FUNCTION_BLOCK FB_A_Magnetventil IMPLEMENTS I_Magnetventil
VAR_INPUT
	I_iModus			:INT;		// Zustand des Systems (z.B. 0 = AUS | 1 = MAN | 2 = AUTO)
	I_bVerriegeln		:BOOL;		// Verriegelte Elemente sind nicht ansteuerbar
END_VAR

VAR_OUTPUT
	O_bAktivieren		:BOOL;		// Ventil wird geöffnet / geschlossen
	O_bStoerung			:BOOL;		// Befindet sich das Element in einem Error
	O_iStoerungID		:INT;		// Anzeigen von Störung über eine INT-Variable
END_VAR

VAR
END_VAR

// Verriegeln des Systems (Element geht in definierten Zustand) -> Ventil wird geschlossen
IF I_bVerriegeln THEN
	O_bAktivieren := FALSE;
END_IF

METHOD M_A_OEFFNEN : BOOL
VAR_INPUT
END_VAR
// EBENE 1: Verriegelung
IF NOT I_bVerriegeln THEN	
	// EBEN 2: AUTO-Modus
		IF I_iModus = 2 THEN
			O_bAktivieren := TRUE;
		END_IF
END_IF

M_A_OEFFNEN := O_bAktivieren;
END_METHOD

METHOD M_A_SCHLIESSEN : BOOL
VAR_INPUT
END_VAR
IF I_iModus = 2 THEN
	O_bAktivieren := FALSE;
END_IF

M_A_SCHLIESSEN := NOT O_bAktivieren;
END_METHOD

METHOD M_M_OEFFNEN : BOOL
VAR_INPUT
END_VAR
// EBENE 1: Verriegelung
IF NOT I_bVerriegeln THEN	
	// EBEN 2: MAN-Modus
		IF I_iModus = 1 THEN
			O_bAktivieren := TRUE;
		END_IF
END_IF

M_M_OEFFNEN := O_bAktivieren;
END_METHOD

METHOD M_M_SCHLIESSEN : BOOL
VAR_INPUT
END_VAR
IF I_iModus = 1 THEN
	O_bAktivieren := FALSE;
END_IF

M_M_SCHLIESSEN := NOT O_bAktivieren;
END_METHOD

PROPERTY P_Status : INT
GET
IF O_bAktivieren THEN
	P_Status := 1;
ELSE
	P_Status := 0;
END_IF
END_GET
END_PROPERTY

END_FUNCTION_BLOCK

(* stored: Version 1.1.0.1, ProductVersion 3.1.4024.12
   POU FB_A_Magnetventil: Id {09d7eebc-a3d6-472d-9daa-768caf665633}, SpecialFunc None
   Method M_A_OEFFNEN: Id {2e1a37fd-2447-4a2a-88c2-4af5bfca4510}
   Method M_A_SCHLIESSEN: Id {635c5620-4889-48ab-b592-2ac4b242d83c}
   Method M_M_OEFFNEN: Id {81ef93b3-6f19-40d1-92ae-bcbddac32bb5}
   Method M_M_SCHLIESSEN: Id {703bd2e7-cfb9-48e5-8885-a164ebac1fc0}
   Property P_Status: Id {e3c7b6b4-46cf-4afc-aa3d-2c467bea2077}
   Get Get: Id {7a240f48-917c-49d2-a9f2-c5d67c2c06f7} *)
